LIN {X 0,Y 119.717,Z 305.18,A -85,B 0,C 180,E1 -30603.649,E2 -30603.649} C_VEL
LIN {X 0,Y 116.126,Z 315.063,A -85,B 0,C 180,E1 -30603.943,E2 -30603.943} C_VEL
LIN {X 0,Y 111.009,Z 325.952,A -85,B 0,C 180,E1 -30604.349,E2 -30604.349} C_VEL
LIN {X 0,Y 105.794,Z 334.941,A -85,B 0,C 180,E1 -30604.827,E2 -30604.827} C_VEL
LIN {X 0,Y 99.722,Z 343.662,A -85,B 0,C 180,E1 -30605.461,E2 -30605.461} C_VEL
LIN {X 0,Y 93.661,Z 351.048,A -85,B 0,C 180,E1 -30606.163,E2 -30606.163} C_VEL
LIN {X 0,Y 86.76,Z 358.26,A -85,B 0,C 180,E1 -30607.115,E2 -30607.115} C_VEL
LIN {X 0,Y 79.892,Z 364.456,A -85,B 0,C 180,E1 -30608.255,E2 -30608.255} C_VEL
LIN {X 0,Y 71.375,Z 370.99,A -85,B 0,C 180,E1 -30610.054,E2 -30610.054} C_VEL
LIN {X 0,Y 64.619,Z 375.489,A -85,B 0,C 180,E1 -30611.811,E2 -30611.811} C_VEL
LIN {X 0,Y 54.695,Z 380.985,A -85,B 0,C 180,E1 -30615.484,E2 -30615.484} C_VEL
LIN {X 0,Y 45.01,Z 385.31,A -85,B 0,C 180,E1 -30620.47,E2 -30620.47} C_VEL
LIN {X 0,Y 38.837,Z 387.682,A -85,B 0,C 180,E1 -30625.205,E2 -30625.205} C_VEL
LIN {X 0,Y 32.984,Z 389.485,A -85,B 0,C 180,E1 -30631.54,E2 -30631.54} C_VEL
LIN {X 0,Y 23.511,Z 391.952,A -85,B 0,C 180,E1 -30653.284,E2 -30653.284} C_VEL
LIN {X 0,Y 20.752,Z 392.553,A -85,B 0,C 180,E1 -30670.204,E2 -30670.204} C_VEL
LIN {X 0,Y 19.969,Z 392.717,A -85,B 0,C 180,E1 -30690,E2 -30690} C_VEL
LIN {X 0,Y 20.693,Z 392.552,A -85,B 0,C 180,E1 -30709.854,E2 -30709.854} C_VEL
LIN {X 0,Y 23.498,Z 391.951,A -85,B 0,C 180,E1 -30726.739,E2 -30726.739} C_VEL
LIN {X 0,Y 32.981,Z 389.485,A -85,B 0,C 180,E1 -30748.468,E2 -30748.468} C_VEL
LIN {X 0,Y 41.901,Z 386.53,A -85,B 0,C 180,E1 -30757.293,E2 -30757.293} C_VEL
LIN {X 0,Y 51.443,Z 382.54,A -85,B 0,C 180,E1 -30763,E2 -30763} C_VEL
LIN {X 0,Y 60.969,Z 377.599,A -85,B 0,C 180,E1 -30766.915,E2 -30766.915} C_VEL
LIN {X 0,Y 69.682,Z 372.145,A -85,B 0,C 180,E1 -30769.533,E2 -30769.533} C_VEL
LIN {X 0,Y 78.182,Z 365.831,A -85,B 0,C 180,E1 -30771.422,E2 -30771.422} C_VEL
LIN {X 0,Y 85.041,Z 359.886,A -85,B 0,C 180,E1 -30772.61,E2 -30772.61} C_VEL
LIN {X 0,Y 91.927,Z 352.964,A -85,B 0,C 180,E1 -30773.652,E2 -30773.652} C_VEL
LIN {X 0,Y 98.848,Z 344.794,A -85,B 0,C 180,E1 -30774.487,E2 -30774.487} C_VEL
LIN {X 0,Y 104.925,Z 336.291,A -85,B 0,C 180,E1 -30775.094,E2 -30775.094} C_VEL
LIN {X 0,Y 110.138,Z 327.582,A -85,B 0,C 180,E1 -30775.587,E2 -30775.587} C_VEL
LIN {X 0,Y 114.838,Z 318.036,A -85,B 0,C 180,E1 -30775.963,E2 -30775.963} C_VEL
LIN {X 0,Y 118.374,Z 309.139,A -85,B 0,C 180,E1 -30776.272,E2 -30776.272} C_VEL
LIN {X 0,Y 119.713,Z 305.178,A -85,B 0,C 180,E1 -30776.385,E2 -30776.385} C_VEL
LIN {X 0,Y 120.248,Z 303.503,A -85,B 0,C 180,E1 -30776.648,E2 -30776.648} C_VEL
LIN {X 0,Y 120.44,Z 302.029,A -85,B 0,C 180,E1 -30779.998,E2 -30779.998} C_VEL
LIN {X 0,Y 120.194,Z 303.28,A -85,B 0,C 180,E1 -30783.35,E2 -30783.35} C_VEL
LIN {X 0,Y 120.067,Z 305.276,A -85,B 0,C 180,E1 -30786.721,E2 -30786.721} C_VEL
LIN {X 0,Y 120.02,Z 306.688,A -85,B 0,C 180,E1 -30788.416,E2 -30788.416} C_VEL
LIN {X 0,Y 119.884,Z 309.705,A -85,B 0,C 180,E1 -30791.086,E2 -30791.086} C_VEL
LIN {X 0,Y 119.455,Z 313.518,A -85,B 0,C 180,E1 -30793.609,E2 -30793.609} C_VEL
LIN {X 0,Y 118.463,Z 318.955,A -85,B 0,C 180,E1 -30796.366,E2 -30796.366} C_VEL
LIN {X 0,Y 115.432,Z 330.435,A -85,B 0,C 180,E1 -30801.424,E2 -30801.424} C_VEL
LIN {X 0,Y 112.841,Z 339.939,A -85,B 0,C 180,E1 -30806.593,E2 -30806.593} C_VEL
LIN {X 0,Y 110.853,Z 348.799,A -85,B 0,C 180,E1 -30812.532,E2 -30812.532} C_VEL
LIN {X 0,Y 109.913,Z 356.079,A -85,B 0,C 180,E1 -30818.394,E2 -30818.394} C_VEL
LIN {X 0,Y 110.102,Z 362.578,A -85,B 0,C 180,E1 -30824.597,E2 -30824.597} C_VEL
LIN {X 0,Y 111.723,Z 368.309,A -85,B 0,C 180,E1 -30831.02,E2 -30831.02} C_VEL
LIN {X 0,Y 115.499,Z 373.969,A -85,B 0,C 180,E1 -30838.413,E2 -30838.413} C_VEL
LIN {X 0,Y 120.451,Z 378.02,A -85,B 0,C 180,E1 -30844.486,E2 -30844.486} C_VEL
LIN {X 0,Y 127.757,Z 381.631,A -85,B 0,C 180,E1 -30850.727,E2 -30850.727} C_VEL
LIN {X 0,Y 137.278,Z 384.47,A -85,B 0,C 180,E1 -30856.578,E2 -30856.578} C_VEL
LIN {X 0,Y 149.17,Z 386.419,A -85,B 0,C 180,E1 -30861.875,E2 -30861.875} C_VEL
LIN {X 0,Y 161.996,Z 387.374,A -85,B 0,C 180,E1 -30866.197,E2 -30866.197} C_VEL
LIN {X 0,Y 176.187,Z 387.451,A -85,B 0,C 180,E1 -30870,E2 -30870} C_VEL
LIN {X 0,Y 161.994,Z 387.377,A -85,B 0,C 180,E1 -30873.788,E2 -30873.788} C_VEL
LIN {X 0,Y 156.857,Z 387.171,A -85,B 0,C 180,E1 -30875.379,E2 -30875.379} C_VEL
LIN {X 0,Y 152.092,Z 386.947,A -85,B 0,C 180,E1 -30876.675,E2 -30876.675} C_VEL
LIN {X 0,Y 136.433,Z 386.309,A -85,B 0,C 180,E1 -30880.073,E2 -30880.073} C_VEL
LIN {X 0,Y 131.842,Z 385.916,A -85,B 0,C 180,E1 -30881.644,E2 -30881.644} C_VEL
LIN {X 0,Y 130.521,Z 385.655,A -85,B 0,C 180,E1 -30882.275,E2 -30882.275} C_VEL
LIN {X 0,Y 123.482,Z 384.041,A -85,B 0,C 180,E1 -30886.533,E2 -30886.533} C_VEL
LIN {X 0,Y 114.992,Z 380.706,A -85,B 0,C 180,E1 -30893.549,E2 -30893.549} C_VEL
LIN {X 0,Y 108.159,Z 375.569,A -85,B 0,C 180,E1 -30902.362,E2 -30902.362} C_VEL
LIN {X 0,Y 104.996,Z 370.6,A -85,B 0,C 180,E1 -30909.671,E2 -30909.671} C_VEL
LIN {X 0,Y 103.683,Z 364.458,A -85,B 0,C 180,E1 -30917.328,E2 -30917.328} C_VEL
LIN {X 0,Y 104.187,Z 357.94,A -85,B 0,C 180,E1 -30924.043,E2 -30924.043} C_VEL
LIN {X 0,Y 105.674,Z 351.257,A -85,B 0,C 180,E1 -30929.834,E2 -30929.834} C_VEL
LIN {X 0,Y 108.139,Z 343.326,A -85,B 0,C 180,E1 -30935.485,E2 -30935.485} C_VEL
LIN {X 0,Y 110.828,Z 335.561,A -85,B 0,C 180,E1 -30940.076,E2 -30940.076} C_VEL
LIN {X 0,Y 114.078,Z 326.223,A -85,B 0,C 180,E1 -30944.597,E2 -30944.597} C_VEL
LIN {X 0,Y 116.107,Z 319.796,A -85,B 0,C 180,E1 -30947.593,E2 -30947.593} C_VEL
LIN {X 0,Y 117.011,Z 315.348,A -85,B 0,C 180,E1 -30950.495,E2 -30950.495} C_VEL
LIN {X 0,Y 117.648,Z 311.793,A -85,B 0,C 180,E1 -30954.051,E2 -30954.051} C_VEL
LIN {X 0,Y 117.816,Z 310.254,A -85,B 0,C 180,E1 -30956.582,E2 -30956.582} C_VEL
LIN {X 0,Y 118.131,Z 308.908,A -85,B 0,C 180,E1 -30960.002,E2 -30960.002} C_VEL
LIN {X 0,Y 117.855,Z 309.739,A -85,B 0,C 180,E1 -30960.319,E2 -30960.319} C_VEL
LIN {X 0,Y 112.453,Z 322.497,A -85,B 0,C 180,E1 -30960.592,E2 -30960.592} C_VEL
LIN {X 0,Y 106.311,Z 333.399,A -85,B 0,C 180,E1 -30960.926,E2 -30960.926} C_VEL
LIN {X 0,Y 100.174,Z 342.337,A -85,B 0,C 180,E1 -30961.31,E2 -30961.31} C_VEL
LIN {X 0,Y 93.166,Z 350.856,A -85,B 0,C 180,E1 -30961.801,E2 -30961.801} C_VEL
LIN {X 0,Y 86.169,Z 358.068,A -85,B 0,C 180,E1 -30962.416,E2 -30962.416} C_VEL
LIN {X 0,Y 79.183,Z 364.264,A -85,B 0,C 180,E1 -30963.146,E2 -30963.146} C_VEL
LIN {X 0,Y 70.481,Z 370.797,A -85,B 0,C 180,E1 -30964.337,E2 -30964.337} C_VEL
LIN {X 0,Y 63.544,Z 375.296,A -85,B 0,C 180,E1 -30965.506,E2 -30965.506} C_VEL
LIN {X 0,Y 54.523,Z 380.204,A -85,B 0,C 180,E1 -30967.657,E2 -30967.657} C_VEL
LIN {X 0,Y 46.422,Z 383.878,A -85,B 0,C 180,E1 -30970.249,E2 -30970.249} C_VEL
LIN {X 0,Y 36.38,Z 387.49,A -85,B 0,C 180,E1 -30975.003,E2 -30975.003} C_VEL
LIN {X 0,Y 29.879,Z 389.292,A -85,B 0,C 180,E1 -30979.807,E2 -30979.807} C_VEL
LIN {X 0,Y 18.307,Z 391.76,A -85,B 0,C 180,E1 -30999.844,E2 -30999.844} C_VEL
LIN {X 0,Y 14.255,Z 392.361,A -85,B 0,C 180,E1 -31020.461,E2 -31020.461} C_VEL
LIN {X 0,Y 12.863,Z 392.526,A -85,B 0,C 180,E1 -31050,E2 -31050} C_VEL
LIN {X 0,Y 14.211,Z 392.36,A -85,B 0,C 180,E1 -31079.64,E2 -31079.64} C_VEL
LIN {X 0,Y 18.298,Z 391.759,A -85,B 0,C 180,E1 -31100.189,E2 -31100.189} C_VEL
LIN {X 0,Y 29.878,Z 389.292,A -85,B 0,C 180,E1 -31120.201,E2 -31120.201} C_VEL
LIN {X 0,Y 39.698,Z 386.338,A -85,B 0,C 180,E1 -31126.825,E2 -31126.825} C_VEL
LIN {X 0,Y 49.826,Z 382.347,A -85,B 0,C 180,E1 -31130.877,E2 -31130.877} C_VEL
LIN {X 0,Y 56.661,Z 379.131,A -85,B 0,C 180,E1 -31132.871,E2 -31132.871} C_VEL
LIN {X 0,Y 67.01,Z 373.107,A -85,B 0,C 180,E1 -31135.098,E2 -31135.098} C_VEL
LIN {X 0,Y 75.698,Z 367.014,A -85,B 0,C 180,E1 -31136.42,E2 -31136.42} C_VEL
LIN {X 0,Y 82.675,Z 361.319,A -85,B 0,C 180,E1 -31137.231,E2 -31137.231} C_VEL
LIN {X 0,Y 91.414,Z 352.772,A -85,B 0,C 180,E1 -31138.084,E2 -31138.084} C_VEL
LIN {X 0,Y 98.42,Z 344.602,A -85,B 0,C 180,E1 -31138.601,E2 -31138.601} C_VEL
LIN {X 0,Y 104.557,Z 336.1,A -85,B 0,C 180,E1 -31138.968,E2 -31138.968} C_VEL
LIN {X 0,Y 109.82,Z 327.39,A -85,B 0,C 180,E1 -31139.289,E2 -31139.289} C_VEL
LIN {X 0,Y 114.558,Z 317.844,A -85,B 0,C 180,E1 -31139.51,E2 -31139.51} C_VEL
LIN {X 0,Y 117.855,Z 309.739,A -85,B 0,C 180,E1 -31139.689,E2 -31139.689} C_VEL
LIN {X 0,Y 118.131,Z 308.909,A -85,B 0,C 180,E1 -31139.998,E2 -31139.998} C_VEL
LIN {X 0,Y 117.815,Z 310.257,A -85,B 0,C 180,E1 -31143.418,E2 -31143.418} C_VEL
LIN {X 0,Y 117.528,Z 312.556,A -85,B 0,C 180,E1 -31146.867,E2 -31146.867} C_VEL
LIN {X 0,Y 117.015,Z 315.34,A -85,B 0,C 180,E1 -31149.505,E2 -31149.505} C_VEL
LIN {X 0,Y 116.112,Z 319.784,A -85,B 0,C 180,E1 -31152.406,E2 -31152.406} C_VEL
LIN {X 0,Y 114.581,Z 324.734,A -85,B 0,C 180,E1 -31154.762,E2 -31154.762} C_VEL
LIN {X 0,Y 111.471,Z 333.723,A -85,B 0,C 180,E1 -31158.966,E2 -31158.966} C_VEL
LIN {X 0,Y 109.082,Z 340.55,A -85,B 0,C 180,E1 -31162.739,E2 -31162.739} C_VEL
LIN {X 0,Y 106.334,Z 349.039,A -85,B 0,C 180,E1 -31168.488,E2 -31168.488} C_VEL
LIN {X 0,Y 104.477,Z 356.334,A -85,B 0,C 180,E1 -31174.467,E2 -31174.467} C_VEL
LIN {X 0,Y 103.688,Z 362.492,A -85,B 0,C 180,E1 -31180.491,E2 -31180.491} C_VEL
LIN {X 0,Y 104.337,Z 368.701,A -85,B 0,C 180,E1 -31187.809,E2 -31187.809} C_VEL
LIN {X 0,Y 106.893,Z 374.031,A -85,B 0,C 180,E1 -31195.263,E2 -31195.263} C_VEL
LIN {X 0,Y 111.223,Z 378.305,A -85,B 0,C 180,E1 -31202.203,E2 -31202.203} C_VEL
LIN {X 0,Y 117.698,Z 381.92,A -85,B 0,C 180,E1 -31209.006,E2 -31209.006} C_VEL
LIN {X 0,Y 124.291,Z 384.232,A -85,B 0,C 180,E1 -31213.992,E2 -31213.992} C_VEL
LIN {X 0,Y 135.506,Z 386.463,A -85,B 0,C 180,E1 -31220.197,E2 -31220.197} C_VEL
LIN {X 0,Y 148.1,Z 387.613,A -85,B 0,C 180,E1 -31225.215,E2 -31225.215} C_VEL
LIN {X 0,Y 164.229,Z 387.768,A -85,B 0,C 180,E1 -31230,E2 -31230} C_VEL
LIN {X 0,Y 148.095,Z 387.618,A -85,B 0,C 180,E1 -31234.764,E2 -31234.764} C_VEL
LIN {X 0,Y 135.506,Z 386.463,A -85,B 0,C 180,E1 -31239.803,E2 -31239.803} C_VEL
LIN {X 0,Y 130.521,Z 385.655,A -85,B 0,C 180,E1 -31242.275,E2 -31242.275} C_VEL
LIN {X 0,Y 126.383,Z 385.107,A -85,B 0,C 180,E1 -31244.144,E2 -31244.144} C_VEL
LIN {X 0,Y 112.702,Z 383.535,A -85,B 0,C 180,E1 -31249.585,E2 -31249.585} C_VEL
LIN {X 0,Y 109.04,Z 382.656,A -85,B 0,C 180,E1 -31251.925,E2 -31251.925} C_VEL
LIN {X 0,Y 108.082,Z 382.289,A -85,B 0,C 180,E1 -31252.809,E2 -31252.809} C_VEL
LIN {X 0,Y 103.628,Z 379.673,A -85,B 0,C 180,E1 -31258.342,E2 -31258.342} C_VEL
LIN {X 0,Y 99.538,Z 375.349,A -85,B 0,C 180,E1 -31266.247,E2 -31266.247} C_VEL
LIN {X 0,Y 97.636,Z 370.393,A -85,B 0,C 180,E1 -31273.964,E2 -31273.964} C_VEL
LIN {X 0,Y 97.46,Z 366.272,A -85,B 0,C 180,E1 -31279.536,E2 -31279.536} C_VEL
LIN {X 0,Y 98.847,Z 359.058,A -85,B 0,C 180,E1 -31287.491,E2 -31287.491} C_VEL
LIN {X 0,Y 100.988,Z 352.866,A -85,B 0,C 180,E1 -31293.11,E2 -31293.11} C_VEL
LIN {X 0,Y 104.52,Z 344.31,A -85,B 0,C 180,E1 -31299.333,E2 -31299.333} C_VEL
LIN {X 0,Y 108.138,Z 335.987,A -85,B 0,C 180,E1 -31304.221,E2 -31304.221} C_VEL
LIN {X 0,Y 111.793,Z 327.342,A -85,B 0,C 180,E1 -31308.347,E2 -31308.347} C_VEL
LIN {X 0,Y 113.197,Z 323.573,A -85,B 0,C 180,E1 -31310.282,E2 -31310.282} C_VEL
LIN {X 0,Y 114.321,Z 319.955,A -85,B 0,C 180,E1 -31312.939,E2 -31312.939} C_VEL
LIN {X 0,Y 114.743,Z 318.21,A -85,B 0,C 180,E1 -31314.73,E2 -31314.73} C_VEL
LIN {X 0,Y 114.98,Z 317.143,A -85,B 0,C 180,E1 -31316.498,E2 -31316.498} C_VEL
LIN {X 0,Y 114.32,Z 318.561,A -85,B 0,C 180,E1 -31316.943,E2 -31316.943} C_VEL
LIN {X 0,Y 108.198,Z 330.439,A -85,B 0,C 180,E1 -31317.047,E2 -31317.047} C_VEL
LIN {X 0,Y 101.146,Z 341.011,A -85,B 0,C 180,E1 -31317.218,E2 -31317.218} C_VEL
LIN {X 0,Y 94.977,Z 348.747,A -85,B 0,C 180,E1 -31317.371,E2 -31317.371} C_VEL
LIN {X 0,Y 86.162,Z 357.876,A -85,B 0,C 180,E1 -31317.688,E2 -31317.688} C_VEL
LIN {X 0,Y 79.113,Z 364.072,A -85,B 0,C 180,E1 -31317.991,E2 -31317.991} C_VEL
LIN {X 0,Y 70.302,Z 370.605,A -85,B 0,C 180,E1 -31318.541,E2 -31318.541} C_VEL
LIN {X 0,Y 63.26,Z 375.104,A -85,B 0,C 180,E1 -31319.06,E2 -31319.06} C_VEL
LIN {X 0,Y 53.07,Z 380.439,A -85,B 0,C 180,E1 -31320.253,E2 -31320.253} C_VEL
LIN {X 0,Y 42.194,Z 384.926,A -85,B 0,C 180,E1 -31322.012,E2 -31322.012} C_VEL
LIN {X 0,Y 35.215,Z 387.298,A -85,B 0,C 180,E1 -31323.744,E2 -31323.744} C_VEL
LIN {X 0,Y 28.272,Z 389.1,A -85,B 0,C 180,E1 -31326.096,E2 -31326.096} C_VEL
LIN {X 0,Y 14.789,Z 391.567,A -85,B 0,C 180,E1 -31338.122,E2 -31338.122} C_VEL
LIN {X 0,Y 8.797,Z 392.169,A -85,B 0,C 180,E1 -31356.976,E2 -31356.976} C_VEL
LIN {X 0,Y 5.749,Z 392.334,A -85,B 0,C 180,E1 -31410,E2 -31410} C_VEL
LIN {X 0,Y 8.772,Z 392.168,A -85,B 0,C 180,E1 -31463.24,E2 -31463.24} C_VEL
LIN {X 0,Y 14.786,Z 391.567,A -85,B 0,C 180,E1 -31481.923,E2 -31481.923} C_VEL
LIN {X 0,Y 28.271,Z 389.1,A -85,B 0,C 180,E1 -31493.912,E2 -31493.912} C_VEL
LIN {X 0,Y 38.701,Z 386.145,A -85,B 0,C 180,E1 -31497.174,E2 -31497.174} C_VEL
LIN {X 0,Y 49.201,Z 382.155,A -85,B 0,C 180,E1 -31499.113,E2 -31499.113} C_VEL
LIN {X 0,Y 56.223,Z 378.938,A -85,B 0,C 180,E1 -31500.109,E2 -31500.109} C_VEL
LIN {X 0,Y 66.78,Z 372.915,A -85,B 0,C 180,E1 -31501.195,E2 -31501.195} C_VEL
LIN {X 0,Y 75.588,Z 366.822,A -85,B 0,C 180,E1 -31501.819,E2 -31501.819} C_VEL
LIN {X 0,Y 82.637,Z 361.127,A -85,B 0,C 180,E1 -31502.16,E2 -31502.16} C_VEL
LIN {X 0,Y 91.453,Z 352.58,A -85,B 0,C 180,E1 -31502.542,E2 -31502.542} C_VEL
LIN {X 0,Y 98.503,Z 344.411,A -85,B 0,C 180,E1 -31502.731,E2 -31502.731} C_VEL
LIN {X 0,Y 104.67,Z 335.908,A -85,B 0,C 180,E1 -31502.852,E2 -31502.852} C_VEL
LIN {X 0,Y 109.73,Z 327.624,A -85,B 0,C 180,E1 -31502.981,E2 -31502.981} C_VEL
LIN {X 0,Y 114.154,Z 318.938,A -85,B 0,C 180,E1 -31503.048,E2 -31503.048} C_VEL
LIN {X 0,Y 114.977,Z 317.151,A -85,B 0,C 180,E1 -31503.502,E2 -31503.502} C_VEL
LIN {X 0,Y 114.73,Z 318.239,A -85,B 0,C 180,E1 -31505.27,E2 -31505.27} C_VEL
LIN {X 0,Y 114.07,Z 320.946,A -85,B 0,C 180,E1 -31507.878,E2 -31507.878} C_VEL
LIN {X 0,Y 113.191,Z 323.583,A -85,B 0,C 180,E1 -31509.718,E2 -31509.718} C_VEL
LIN {X 0,Y 111.794,Z 327.348,A -85,B 0,C 180,E1 -31511.664,E2 -31511.664} C_VEL
LIN {X 0,Y 107.515,Z 337.525,A -85,B 0,C 180,E1 -31516.593,E2 -31516.593} C_VEL
LIN {X 0,Y 103.001,Z 347.918,A -85,B 0,C 180,E1 -31523.097,E2 -31523.097} C_VEL
LIN {X 0,Y 99.626,Z 356.578,A -85,B 0,C 180,E1 -31530.163,E2 -31530.163} C_VEL
LIN {X 0,Y 97.918,Z 362.751,A -85,B 0,C 180,E1 -31536.37,E2 -31536.37} C_VEL
LIN {X 0,Y 97.425,Z 368.832,A -85,B 0,C 180,E1 -31543.832,E2 -31543.832} C_VEL
LIN {X 0,Y 98.753,Z 374.021,A -85,B 0,C 180,E1 -31551.518,E2 -31551.518} C_VEL
LIN {X 0,Y 102.11,Z 378.453,A -85,B 0,C 180,E1 -31559.266,E2 -31559.266} C_VEL
LIN {X 0,Y 107.875,Z 382.206,A -85,B 0,C 180,E1 -31566.99,E2 -31566.99} C_VEL
LIN {X 0,Y 113.233,Z 384.33,A -85,B 0,C 180,E1 -31571.921,E2 -31571.921} C_VEL
LIN {X 0,Y 122.133,Z 386.449,A -85,B 0,C 180,E1 -31578.018,E2 -31578.018} C_VEL
LIN {X 0,Y 134.476,Z 387.839,A -85,B 0,C 180,E1 -31584,E2 -31584} C_VEL
LIN {X 0,Y 147.626,Z 388.209,A -85,B 0,C 180,E1 -31588.622,E2 -31588.622} C_VEL
LIN {X 0,Y 152.296,Z 388.084,A -85,B 0,C 180,E1 -31590,E2 -31590} C_VEL
LIN {X 0,Y 140.828,Z 388.098,A -85,B 0,C 180,E1 -31593.564,E2 -31593.564} C_VEL
LIN {X 0,Y 128.019,Z 387.219,A -85,B 0,C 180,E1 -31598.836,E2 -31598.836} C_VEL
LIN {X 0,Y 119.391,Z 385.888,A -85,B 0,C 180,E1 -31603.619,E2 -31603.619} C_VEL
LIN {X 0,Y 111.723,Z 383.815,A -85,B 0,C 180,E1 -31609.344,E2 -31609.344} C_VEL
LIN {X 0,Y 108.082,Z 382.289,A -85,B 0,C 180,E1 -31612.809,E2 -31612.809} C_VEL
LIN {X 0,Y 105.046,Z 381.281,A -85,B 0,C 180,E1 -31615.486,E2 -31615.486} C_VEL
LIN {X 0,Y 94.843,Z 378.641,A -85,B 0,C 180,E1 -31623.749,E2 -31623.749} C_VEL
LIN {X 0,Y 92.636,Z 377.218,A -85,B 0,C 180,E1 -31626.968,E2 -31626.968} C_VEL
LIN {X 0,Y 92.209,Z 376.621,A -85,B 0,C 180,E1 -31628.096,E2 -31628.096} C_VEL
LIN {X 0,Y 91.002,Z 372.12,A -85,B 0,C 180,E1 -31635.971,E2 -31635.971} C_VEL
LIN {X 0,Y 91.937,Z 365.634,A -85,B 0,C 180,E1 -31645.023,E2 -31645.023} C_VEL
LIN {X 0,Y 94.304,Z 359.218,A -85,B 0,C 180,E1 -31652.244,E2 -31652.244} C_VEL
LIN {X 0,Y 97.979,Z 351.735,A -85,B 0,C 180,E1 -31658.824,E2 -31658.824} C_VEL
LIN {X 0,Y 102.175,Z 343.794,A -85,B 0,C 180,E1 -31664.357,E2 -31664.357} C_VEL
LIN {X 0,Y 106.125,Z 336.294,A -85,B 0,C 180,E1 -31668.543,E2 -31668.543} C_VEL
LIN {X 0,Y 109.814,Z 328.832,A -85,B 0,C 180,E1 -31672.195,E2 -31672.195} C_VEL
LIN {X 0,Y 110.156,Z 328.004,A -85,B 0,C 180,E1 -31672.671,E2 -31672.671} C_VEL
LIN {X 0,Y 109.108,Z 329.688,A -85,B 0,C 180,E1 -31673.32,E2 -31673.32} C_VEL
LIN {X 0,Y 101.739,Z 340.819,A -85,B 0,C 180,E1 -31673.215,E2 -31673.215} C_VEL
LIN {X 0,Y 95.565,Z 348.556,A -85,B 0,C 180,E1 -31673.121,E2 -31673.121} C_VEL
LIN {X 0,Y 86.741,Z 357.685,A -85,B 0,C 180,E1 -31672.988,E2 -31672.988} C_VEL
LIN {X 0,Y 79.682,Z 363.879,A -85,B 0,C 180,E1 -31672.862,E2 -31672.862} C_VEL
LIN {X 0,Y 70.844,Z 370.412,A -85,B 0,C 180,E1 -31672.759,E2 -31672.759} C_VEL
LIN {X 0,Y 63.775,Z 374.912,A -85,B 0,C 180,E1 -31672.652,E2 -31672.652} C_VEL
LIN {X 0,Y 52.528,Z 380.681,A -85,B 0,C 180,E1 -31672.569,E2 -31672.569} C_VEL
LIN {X 0,Y 42.543,Z 384.734,A -85,B 0,C 180,E1 -31672.384,E2 -31672.384} C_VEL
LIN {X 0,Y 35.468,Z 387.105,A -85,B 0,C 180,E1 -31672.192,E2 -31672.192} C_VEL
LIN {X 0,Y 28.411,Z 388.908,A -85,B 0,C 180,E1 -31671.673,E2 -31671.673} C_VEL
LIN {X 0,Y 14.284,Z 391.375,A -85,B 0,C 180,E1 -31669.74,E2 -31669.74} C_VEL
LIN {X 0,Y 7.265,Z 391.977,A -85,B 0,C 180,E1 -31665.323,E2 -31665.323} C_VEL
LIN {X 0,Y 1.35,Z 392.142,A -85,B 0,C 180,E1 -31590,E2 -31590} C_VEL
LIN {X 0,Y 7.274,Z 391.976,A -85,B 0,C 180,E1 -31514.953,E2 -31514.953} C_VEL
LIN {X 0,Y 14.286,Z 391.374,A -85,B 0,C 180,E1 -31510.308,E2 -31510.308} C_VEL
LIN {X 0,Y 28.412,Z 388.908,A -85,B 0,C 180,E1 -31508.334,E2 -31508.334} C_VEL
LIN {X 0,Y 39.007,Z 385.952,A -85,B 0,C 180,E1 -31507.723,E2 -31507.723} C_VEL
LIN {X 0,Y 49.607,Z 381.962,A -85,B 0,C 180,E1 -31507.386,E2 -31507.386} C_VEL
LIN {X 0,Y 56.686,Z 378.746,A -85,B 0,C 180,E1 -31507.326,E2 -31507.326} C_VEL
LIN {X 0,Y 67.307,Z 372.723,A -85,B 0,C 180,E1 -31507.272,E2 -31507.272} C_VEL
LIN {X 0,Y 76.147,Z 366.63,A -85,B 0,C 180,E1 -31507.181,E2 -31507.181} C_VEL
LIN {X 0,Y 83.208,Z 360.935,A -85,B 0,C 180,E1 -31507.057,E2 -31507.057} C_VEL
LIN {X 0,Y 92.043,Z 352.388,A -85,B 0,C 180,E1 -31506.967,E2 -31506.967} C_VEL
LIN {X 0,Y 99.095,Z 344.219,A -85,B 0,C 180,E1 -31506.832,E2 -31506.832} C_VEL
LIN {X 0,Y 105.262,Z 335.717,A -85,B 0,C 180,E1 -31506.714,E2 -31506.714} C_VEL
LIN {X 0,Y 109.111,Z 329.682,A -85,B 0,C 180,E1 -31506.68,E2 -31506.68} C_VEL
LIN {X 0,Y 110.169,Z 327.98,A -85,B 0,C 180,E1 -31507.328,E2 -31507.328} C_VEL
LIN {X 0,Y 108.09,Z 332.431,A -85,B 0,C 180,E1 -31509.585,E2 -31509.585} C_VEL
LIN {X 0,Y 103.81,Z 340.756,A -85,B 0,C 180,E1 -31513.814,E2 -31513.814} C_VEL
LIN {X 0,Y 99.099,Z 349.573,A -85,B 0,C 180,E1 -31519.518,E2 -31519.518} C_VEL
LIN {X 0,Y 95.415,Z 356.863,A -85,B 0,C 180,E1 -31525.544,E2 -31525.544} C_VEL
LIN {X 0,Y 92.705,Z 363.199,A -85,B 0,C 180,E1 -31532.048,E2 -31532.048} C_VEL
LIN {X 0,Y 91.098,Z 369.089,A -85,B 0,C 180,E1 -31539.514,E2 -31539.514} C_VEL
LIN {X 0,Y 91.275,Z 374.177,A -85,B 0,C 180,E1 -31547.501,E2 -31547.501} C_VEL
LIN {X 0,Y 93.465,Z 378.582,A -85,B 0,C 180,E1 -31555.801,E2 -31555.801} C_VEL
LIN {X 0,Y 98.43,Z 382.485,A -85,B 0,C 180,E1 -31564.634,E2 -31564.634} C_VEL
LIN {X 0,Y 104.076,Z 384.887,A -85,B 0,C 180,E1 -31570.969,E2 -31570.969} C_VEL
LIN {X 0,Y 114.583,Z 387.2,A -85,B 0,C 180,E1 -31578.911,E2 -31578.911} C_VEL
LIN {X 0,Y 123.062,Z 388.144,A -85,B 0,C 180,E1 -31583.442,E2 -31583.442} C_VEL
LIN {X 0,Y 133.633,Z 388.548,A -85,B 0,C 180,E1 -31587.723,E2 -31587.723} C_VEL
LIN {X 0,Y 140.418,Z 388.398,A -85,B 0,C 180,E1 -31590,E2 -31590} C_VEL
LIN {X 0,Y 126.954,Z 388.307,A -85,B 0,C 180,E1 -31594.85,E2 -31594.85} C_VEL
LIN {X 0,Y 115.539,Z 387.328,A -85,B 0,C 180,E1 -31600.514,E2 -31600.514} C_VEL
LIN {X 0,Y 108.852,Z 386.181,A -85,B 0,C 180,E1 -31604.967,E2 -31604.967} C_VEL
LIN {X 0,Y 101.85,Z 384.071,A -85,B 0,C 180,E1 -31611.281,E2 -31611.281} C_VEL
LIN {X 0,Y 96.204,Z 381.129,A -85,B 0,C 180,E1 -31618.765,E2 -31618.765} C_VEL
LIN {X 0,Y 92.209,Z 376.621,A -85,B 0,C 180,E1 -31628.096,E2 -31628.096} C_VEL
LIN {X 0,Y 90.813,Z 374.958,A -85,B 0,C 180,E1 -31631.533,E2 -31631.533} C_VEL
LIN {X 0,Y 86.018,Z 370.75,A -85,B 0,C 180,E1 -31642.321,E2 -31642.321} C_VEL
LIN {X 0,Y 85.83,Z 368.79,A -85,B 0,C 180,E1 -31646.016,E2 -31646.016} C_VEL
LIN {X 0,Y 86.075,Z 368.012,A -85,B 0,C 180,E1 -31647.204,E2 -31647.204} C_VEL
LIN {X 0,Y 89.354,Z 361.507,A -85,B 0,C 180,E1 -31655.215,E2 -31655.215} C_VEL
LIN {X 0,Y 94.335,Z 353.36,A -85,B 0,C 180,E1 -31662.665,E2 -31662.665} C_VEL
LIN {X 0,Y 99.436,Z 345.305,A -85,B 0,C 180,E1 -31668.306,E2 -31668.306} C_VEL
LIN {X 0,Y 100.182,Z 344.028,A -85,B 0,C 180,E1 -31669.149,E2 -31669.149} C_VEL
LIN {X 0,Y 93.169,Z 352.197,A -85,B 0,C 180,E1 -31668.701,E2 -31668.701} C_VEL
LIN {X 0,Y 84.383,Z 360.743,A -85,B 0,C 180,E1 -31668.127,E2 -31668.127} C_VEL
LIN {X 0,Y 73.843,Z 369.065,A -85,B 0,C 180,E1 -31667.298,E2 -31667.298} C_VEL
LIN {X 0,Y 65.071,Z 374.719,A -85,B 0,C 180,E1 -31666.416,E2 -31666.416} C_VEL
LIN {X 0,Y 54.975,Z 380.018,A -85,B 0,C 180,E1 -31665.19,E2 -31665.19} C_VEL
LIN {X 0,Y 47.521,Z 383.301,A -85,B 0,C 180,E1 -31664.005,E2 -31664.005} C_VEL
LIN {X 0,Y 37.118,Z 386.913,A -85,B 0,C 180,E1 -31661.207,E2 -31661.207} C_VEL
LIN {X 0,Y 23.547,Z 390.111,A -85,B 0,C 180,E1 -31653.559,E2 -31653.559} C_VEL
LIN {X 0,Y 17.068,Z 391.182,A -85,B 0,C 180,E1 -31645.44,E2 -31645.44} C_VEL
LIN {X 0,Y 11.391,Z 391.784,A -85,B 0,C 180,E1 -31628.095,E2 -31628.095} C_VEL
LIN {X 0,Y 8.44,Z 391.951,A -85,B 0,C 180,E1 -31590,E2 -31590} C_VEL
LIN {X 0,Y 11.415,Z 391.784,A -85,B 0,C 180,E1 -31551.998,E2 -31551.998} C_VEL
LIN {X 0,Y 17.074,Z 391.182,A -85,B 0,C 180,E1 -31534.59,E2 -31534.59} C_VEL
LIN {X 0,Y 30.272,Z 388.716,A -85,B 0,C 180,E1 -31521.775,E2 -31521.775} C_VEL
LIN {X 0,Y 40.589,Z 385.759,A -85,B 0,C 180,E1 -31517.766,E2 -31517.766} C_VEL
LIN {X 0,Y 51.023,Z 381.769,A -85,B 0,C 180,E1 -31515.383,E2 -31515.383} C_VEL
LIN {X 0,Y 61.544,Z 376.637,A -85,B 0,C 180,E1 -31513.916,E2 -31513.916} C_VEL
LIN {X 0,Y 70.329,Z 371.376,A -85,B 0,C 180,E1 -31513.016,E2 -31513.016} C_VEL
LIN {X 0,Y 79.118,Z 365.062,A -85,B 0,C 180,E1 -31512.283,E2 -31512.283} C_VEL
LIN {X 0,Y 86.143,Z 359.117,A -85,B 0,C 180,E1 -31511.759,E2 -31511.759} C_VEL
LIN {X 0,Y 93.172,Z 352.197,A -85,B 0,C 180,E1 -31511.308,E2 -31511.308} C_VEL
LIN {X 0,Y 100.187,Z 344.028,A -85,B 0,C 180,E1 -31510.865,E2 -31510.865} C_VEL
LIN {X 0,Y 94.275,Z 353.429,A -85,B 0,C 180,E1 -31517.347,E2 -31517.347} C_VEL
LIN {X 0,Y 89.36,Z 361.514,A -85,B 0,C 180,E1 -31524.807,E2 -31524.807} C_VEL
LIN {X 0,Y 85.841,Z 368.487,A -85,B 0,C 180,E1 -31533.43,E2 -31533.43} C_VEL
LIN {X 0,Y 84.489,Z 373.713,A -85,B 0,C 180,E1 -31541.714,E2 -31541.714} C_VEL
LIN {X 0,Y 85.329,Z 378.598,A -85,B 0,C 180,E1 -31551.477,E2 -31551.477} C_VEL
LIN {X 0,Y 88.672,Z 382.363,A -85,B 0,C 180,E1 -31560.668,E2 -31560.668} C_VEL
LIN {X 0,Y 93.38,Z 384.901,A -85,B 0,C 180,E1 -31567.895,E2 -31567.895} C_VEL
LIN {X 0,Y 101.461,Z 387.121,A -85,B 0,C 180,E1 -31575.863,E2 -31575.863} C_VEL
LIN {X 0,Y 113.189,Z 388.499,A -85,B 0,C 180,E1 -31583.421,E2 -31583.421} C_VEL
LIN {X 0,Y 126.512,Z 388.767,A -85,B 0,C 180,E1 -31589.19,E2 -31589.19} C_VEL
LIN {X 0,Y 128.789,Z 388.706,A -85,B 0,C 180,E1 -31590,E2 -31590} C_VEL
LIN {X 0,Y 119.693,Z 388.782,A -85,B 0,C 180,E1 -31593.48,E2 -31593.48} C_VEL
LIN {X 0,Y 107.072,Z 387.937,A -85,B 0,C 180,E1 -31600.092,E2 -31600.092} C_VEL
LIN {X 0,Y 98.641,Z 386.467,A -85,B 0,C 180,E1 -31606.558,E2 -31606.558} C_VEL
LIN {X 0,Y 92.13,Z 384.353,A -85,B 0,C 180,E1 -31613.743,E2 -31613.743} C_VEL
LIN {X 0,Y 86.397,Z 380.217,A -85,B 0,C 180,E1 -31624.709,E2 -31624.709} C_VEL
LIN {X 0,Y 84.759,Z 377.125,A -85,B 0,C 180,E1 -31631.737,E2 -31631.737} C_VEL
LIN {X 0,Y 84.803,Z 371.698,A -85,B 0,C 180,E1 -31641.658,E2 -31641.658} C_VEL
LIN {X 0,Y 86.075,Z 368.012,A -85,B 0,C 180,E1 -31647.204,E2 -31647.204} C_VEL
LIN {X 0,Y 86.264,Z 366.612,A -85,B 0,C 180,E1 -31649.695,E2 -31649.695} C_VEL
LIN {X 0,Y 85.17,Z 363.237,A -85,B 0,C 180,E1 -31658.412,E2 -31658.412} C_VEL
LIN {X 0,Y 86.09,Z 361.606,A -85,B 0,C 180,E1 -31660.754,E2 -31660.754} C_VEL
LIN {X 0,Y 88.04,Z 358.909,A -85,B 0,C 180,E1 -31663.32,E2 -31663.32} C_VEL
LIN {X 0,Y 87.871,Z 358.925,A -85,B 0,C 180,E1 -31663.691,E2 -31663.691} C_VEL
LIN {X 0,Y 80.931,Z 364.87,A -85,B 0,C 180,E1 -31662.79,E2 -31662.79} C_VEL
LIN {X 0,Y 72.273,Z 371.183,A -85,B 0,C 180,E1 -31661.461,E2 -31661.461} C_VEL
LIN {X 0,Y 63.662,Z 376.443,A -85,B 0,C 180,E1 -31659.778,E2 -31659.778} C_VEL
LIN {X 0,Y 53.373,Z 381.575,A -85,B 0,C 180,E1 -31657.179,E2 -31657.179} C_VEL
LIN {X 0,Y 43.303,Z 385.567,A -85,B 0,C 180,E1 -31653.205,E2 -31653.205} C_VEL
LIN {X 0,Y 33.563,Z 388.524,A -85,B 0,C 180,E1 -31646.884,E2 -31646.884} C_VEL
LIN {X 0,Y 21.913,Z 390.99,A -85,B 0,C 180,E1 -31629.899,E2 -31629.899} C_VEL
LIN {X 0,Y 17.548,Z 391.592,A -85,B 0,C 180,E1 -31613.609,E2 -31613.609} C_VEL
LIN {X 0,Y 15.549,Z 391.759,A -85,B 0,C 180,E1 -31590,E2 -31590} C_VEL
LIN {X 0,Y 17.571,Z 391.592,A -85,B 0,C 180,E1 -31566.423,E2 -31566.423} C_VEL
LIN {X 0,Y 21.921,Z 390.989,A -85,B 0,C 180,E1 -31550.117,E2 -31550.117} C_VEL
LIN {X 0,Y 33.565,Z 388.524,A -85,B 0,C 180,E1 -31533.119,E2 -31533.119} C_VEL
LIN {X 0,Y 43.302,Z 385.567,A -85,B 0,C 180,E1 -31526.792,E2 -31526.792} C_VEL
LIN {X 0,Y 53.364,Z 381.576,A -85,B 0,C 180,E1 -31522.797,E2 -31522.797} C_VEL
LIN {X 0,Y 63.64,Z 376.444,A -85,B 0,C 180,E1 -31520.171,E2 -31520.171} C_VEL
LIN {X 0,Y 72.272,Z 371.183,A -85,B 0,C 180,E1 -31518.538,E2 -31518.538} C_VEL
LIN {X 0,Y 80.929,Z 364.87,A -85,B 0,C 180,E1 -31517.207,E2 -31517.207} C_VEL
LIN {X 0,Y 87.868,Z 358.925,A -85,B 0,C 180,E1 -31516.303,E2 -31516.303} C_VEL
LIN {X 0,Y 88.026,Z 358.91,A -85,B 0,C 180,E1 -31516.652,E2 -31516.652} C_VEL
LIN {X 0,Y 83.121,Z 365.656,A -85,B 0,C 180,E1 -31523.958,E2 -31523.958} C_VEL
LIN {X 0,Y 79.665,Z 371.274,A -85,B 0,C 180,E1 -31531.956,E2 -31531.956} C_VEL
LIN {X 0,Y 77.903,Z 376.343,A -85,B 0,C 180,E1 -31541.381,E2 -31541.381} C_VEL
LIN {X 0,Y 78.466,Z 380.484,A -85,B 0,C 180,E1 -31551.174,E2 -31551.174} C_VEL
LIN {X 0,Y 81.173,Z 383.52,A -85,B 0,C 180,E1 -31559.969,E2 -31559.969} C_VEL
LIN {X 0,Y 84.514,Z 385.4,A -85,B 0,C 180,E1 -31566.162,E2 -31566.162} C_VEL
LIN {X 0,Y 88.793,Z 386.824,A -85,B 0,C 180,E1 -31571.76,E2 -31571.76} C_VEL
LIN {X 0,Y 101.121,Z 388.741,A -85,B 0,C 180,E1 -31582.01,E2 -31582.01} C_VEL
LIN {X 0,Y 112.511,Z 389.144,A -85,B 0,C 180,E1 -31588.022,E2 -31588.022} C_VEL
LIN {X 0,Y 117.26,Z 389.014,A -85,B 0,C 180,E1 -31590,E2 -31590} C_VEL
LIN {X 0,Y 105.85,Z 388.97,A -85,B 0,C 180,E1 -31595.19,E2 -31595.19} C_VEL
LIN {X 0,Y 99.601,Z 388.648,A -85,B 0,C 180,E1 -31598.953,E2 -31598.953} C_VEL
LIN {X 0,Y 88.557,Z 386.753,A -85,B 0,C 180,E1 -31608.508,E2 -31608.508} C_VEL
LIN {X 0,Y 83.999,Z 385.176,A -85,B 0,C 180,E1 -31614.729,E2 -31614.729} C_VEL
LIN {X 0,Y 78.94,Z 381.288,A -85,B 0,C 180,E1 -31626.754,E2 -31626.754} C_VEL
LIN {X 0,Y 77.906,Z 376.348,A -85,B 0,C 180,E1 -31638.604,E2 -31638.604} C_VEL
LIN {X 0,Y 79.375,Z 371.965,A -85,B 0,C 180,E1 -31646.89,E2 -31646.89} C_VEL
LIN {X 0,Y 83.061,Z 365.7,A -85,B 0,C 180,E1 -31656.041,E2 -31656.041} C_VEL
LIN {X 0,Y 86.09,Z 361.606,A -85,B 0,C 180,E1 -31660.754,E2 -31660.754} C_VEL
LIN {X 0,Y 85.175,Z 362.334,A -85,B 0,C 180,E1 -31660.763,E2 -31660.763} C_VEL
LIN {X 0,Y 81.425,Z 365.959,A -85,B 0,C 180,E1 -31658.536,E2 -31658.536} C_VEL
LIN {X 0,Y 75.131,Z 372.49,A -85,B 0,C 180,E1 -31651.444,E2 -31651.444} C_VEL
LIN {X 0,Y 72.376,Z 375.919,A -85,B 0,C 180,E1 -31645.688,E2 -31645.688} C_VEL
LIN {X 0,Y 71.862,Z 376.917,A -85,B 0,C 180,E1 -31643.589,E2 -31643.589} C_VEL
LIN {X 0,Y 71.148,Z 380.747,A -85,B 0,C 180,E1 -31633.745,E2 -31633.745} C_VEL
LIN {X 0,Y 72.252,Z 383.302,A -85,B 0,C 180,E1 -31625.705,E2 -31625.705} C_VEL
LIN {X 0,Y 74.872,Z 385.451,A -85,B 0,C 180,E1 -31617.991,E2 -31617.991} C_VEL
LIN {X 0,Y 81.17,Z 387.695,A -85,B 0,C 180,E1 -31607.755,E2 -31607.755} C_VEL
LIN {X 0,Y 92.177,Z 389.128,A -85,B 0,C 180,E1 -31597.634,E2 -31597.634} C_VEL
LIN {X 0,Y 98.587,Z 389.435,A -85,B 0,C 180,E1 -31593.641,E2 -31593.641} C_VEL
LIN {X 0,Y 105.975,Z 389.318,A -85,B 0,C 180,E1 -31590,E2 -31590} C_VEL
LIN {X 0,Y 97.797,Z 389.394,A -85,B 0,C 180,E1 -31585.879,E2 -31585.879} C_VEL
LIN {X 0,Y 86.326,Z 388.559,A -85,B 0,C 180,E1 -31577.662,E2 -31577.662} C_VEL
LIN {X 0,Y 78.831,Z 387.032,A -85,B 0,C 180,E1 -31569.108,E2 -31569.108} C_VEL
LIN {X 0,Y 73.682,Z 384.681,A -85,B 0,C 180,E1 -31559.137,E2 -31559.137} C_VEL
LIN {X 0,Y 71.704,Z 382.565,A -85,B 0,C 180,E1 -31551.634,E2 -31551.634} C_VEL
LIN {X 0,Y 71.555,Z 377.746,A -85,B 0,C 180,E1 -31538.211,E2 -31538.211} C_VEL
LIN {X 0,Y 74.837,Z 372.04,A -85,B 0,C 180,E1 -31526.857,E2 -31526.857} C_VEL
LIN {X 0,Y 76.535,Z 369.835,A -85,B 0,C 180,E1 -31523.326,E2 -31523.326} C_VEL
LIN {X 0,Y 69.791,Z 374.336,A -85,B 0,C 180,E1 -31525.001,E2 -31525.001} C_VEL
LIN {X 0,Y 58.76,Z 380.319,A -85,B 0,C 180,E1 -31528.578,E2 -31528.578} C_VEL
LIN {X 0,Y 50.059,Z 384.158,A -85,B 0,C 180,E1 -31532.611,E2 -31532.611} C_VEL
LIN {X 0,Y 43.865,Z 386.527,A -85,B 0,C 180,E1 -31536.766,E2 -31536.766} C_VEL
LIN {X 0,Y 37.939,Z 388.332,A -85,B 0,C 180,E1 -31542.186,E2 -31542.186} C_VEL
LIN {X 0,Y 27.763,Z 390.797,A -85,B 0,C 180,E1 -31559.584,E2 -31559.584} C_VEL
LIN {X 0,Y 24.276,Z 391.399,A -85,B 0,C 180,E1 -31573.172,E2 -31573.172} C_VEL
LIN {X 0,Y 22.647,Z 391.567,A -85,B 0,C 180,E1 -31590,E2 -31590} C_VEL
LIN {X 0,Y 24.256,Z 391.4,A -85,B 0,C 180,E1 -31606.842,E2 -31606.842} C_VEL
LIN {X 0,Y 27.755,Z 390.797,A -85,B 0,C 180,E1 -31620.426,E2 -31620.426} C_VEL
LIN {X 0,Y 37.938,Z 388.332,A -85,B 0,C 180,E1 -31637.816,E2 -31637.816} C_VEL
LIN {X 0,Y 46.948,Z 385.374,A -85,B 0,C 180,E1 -31645.419,E2 -31645.419} C_VEL
LIN {X 0,Y 56.527,Z 381.383,A -85,B 0,C 180,E1 -31650.493,E2 -31650.493} C_VEL
LIN {X 0,Y 66.466,Z 376.25,A -85,B 0,C 180,E1 -31653.996,E2 -31653.996} C_VEL
LIN {X 0,Y 73.152,Z 372.146,A -85,B 0,C 180,E1 -31655.88,E2 -31655.88} C_VEL
LIN {X 0,Y 76.171,Z 370.305,A -85,B 0,C 180,E1 -31655.895,E2 -31655.895} C_VEL
LIN {X 0,Y 72.469,Z 375.65,A -85,B 0,C 180,E1 -31646.303,E2 -31646.303} C_VEL
LIN {X 0,Y 71.862,Z 376.917,A -85,B 0,C 180,E1 -31643.589,E2 -31643.589} C_VEL
LIN {X 0,Y 70.647,Z 379.031,A -85,B 0,C 180,E1 -31639.241,E2 -31639.241} C_VEL
LIN {X 0,Y 67.869,Z 382.439,A -85,B 0,C 180,E1 -31631.864,E2 -31631.864} C_VEL
LIN {X 0,Y 66.383,Z 385.181,A -85,B 0,C 180,E1 -31623.88,E2 -31623.88} C_VEL
LIN {X 0,Y 67.21,Z 386.299,A -85,B 0,C 180,E1 -31618.996,E2 -31618.996} C_VEL
LIN {X 0,Y 73.994,Z 388.48,A -85,B 0,C 180,E1 -31606.555,E2 -31606.555} C_VEL
LIN {X 0,Y 79.954,Z 389.319,A -85,B 0,C 180,E1 -31600.125,E2 -31600.125} C_VEL
LIN {X 0,Y 91.407,Z 389.713,A -85,B 0,C 180,E1 -31591.848,E2 -31591.848} C_VEL
LIN {X 0,Y 94.853,Z 389.619,A -85,B 0,C 180,E1 -31590,E2 -31590} C_VEL
LIN {X 0,Y 84.814,Z 389.585,A -85,B 0,C 180,E1 -31583.891,E2 -31583.891} C_VEL
LIN {X 0,Y 78.803,Z 389.242,A -85,B 0,C 180,E1 -31578.808,E2 -31578.808} C_VEL
LIN {X 0,Y 69.286,Z 387.267,A -85,B 0,C 180,E1 -31565.902,E2 -31565.902} C_VEL
LIN {X 0,Y 65.191,Z 384.736,A -85,B 0,C 180,E1 -31553.833,E2 -31553.833} C_VEL
LIN {X 0,Y 64.487,Z 381.173,A -85,B 0,C 180,E1 -31540.832,E2 -31540.832} C_VEL
LIN {X 0,Y 65.56,Z 378.915,A -85,B 0,C 180,E1 -31534.139,E2 -31534.139} C_VEL
LIN {X 0,Y 61.747,Z 380.492,A -85,B 0,C 180,E1 -31534.683,E2 -31534.683} C_VEL
LIN {X 0,Y 54.227,Z 383.966,A -85,B 0,C 180,E1 -31538.958,E2 -31538.958} C_VEL
LIN {X 0,Y 48.478,Z 386.334,A -85,B 0,C 180,E1 -31543.544,E2 -31543.544} C_VEL
LIN {X 0,Y 43.055,Z 388.139,A -85,B 0,C 180,E1 -31549.238,E2 -31549.238} C_VEL
LIN {X 0,Y 34.108,Z 390.605,A -85,B 0,C 180,E1 -31565.663,E2 -31565.663} C_VEL
LIN {X 0,Y 31.161,Z 391.207,A -85,B 0,C 180,E1 -31576.966,E2 -31576.966} C_VEL
LIN {X 0,Y 29.763,Z 391.375,A -85,B 0,C 180,E1 -31590,E2 -31590} C_VEL
LIN {X 0,Y 31.143,Z 391.208,A -85,B 0,C 180,E1 -31603.042,E2 -31603.042} C_VEL
LIN {X 0,Y 34.1,Z 390.605,A -85,B 0,C 180,E1 -31614.342,E2 -31614.342} C_VEL
LIN {X 0,Y 43.054,Z 388.139,A -85,B 0,C 180,E1 -31630.763,E2 -31630.763} C_VEL
LIN {X 0,Y 51.325,Z 385.182,A -85,B 0,C 180,E1 -31638.861,E2 -31638.861} C_VEL
LIN {X 0,Y 60.363,Z 381.19,A -85,B 0,C 180,E1 -31644.587,E2 -31644.587} C_VEL
LIN {X 0,Y 61.39,Z 380.683,A -85,B 0,C 180,E1 -31645.087,E2 -31645.087} C_VEL
LIN {X 0,Y 65.572,Z 378.912,A -85,B 0,C 180,E1 -31645.858,E2 -31645.858} C_VEL
LIN {X 0,Y 64.346,Z 382.502,A -85,B 0,C 180,E1 -31634.981,E2 -31634.981} C_VEL
LIN {X 0,Y 66.245,Z 385.745,A -85,B 0,C 180,E1 -31621.933,E2 -31621.933} C_VEL
LIN {X 0,Y 67.21,Z 386.299,A -85,B 0,C 180,E1 -31618.996,E2 -31618.996} C_VEL
LIN {X 0,Y 68.554,Z 387.366,A -85,B 0,C 180,E1 -31614.199,E2 -31614.199} C_VEL
LIN {X 0,Y 70.205,Z 388.825,A -85,B 0,C 180,E1 -31606.201,E2 -31606.201} C_VEL
LIN {X 0,Y 72.43,Z 389.628,A -85,B 0,C 180,E1 -31600.133,E2 -31600.133} C_VEL
LIN {X 0,Y 75.326,Z 389.924,A -85,B 0,C 180,E1 -31596.169,E2 -31596.169} C_VEL
LIN {X 0,Y 76.586,Z 389.992,A -85,B 0,C 180,E1 -31595.037,E2 -31595.037} C_VEL
LIN {X 0,Y 83.889,Z 389.915,A -85,B 0,C 180,E1 -31590,E2 -31590} C_VEL
LIN {X 0,Y 76.28,Z 389.976,A -85,B 0,C 180,E1 -31584.714,E2 -31584.714} C_VEL
LIN {X 0,Y 65.944,Z 389.092,A -85,B 0,C 180,E1 -31573.561,E2 -31573.561} C_VEL
LIN {X 0,Y 60.324,Z 387.579,A -85,B 0,C 180,E1 -31562.224,E2 -31562.224} C_VEL
LIN {X 0,Y 57.526,Z 384.791,A -85,B 0,C 180,E1 -31547.135,E2 -31547.135} C_VEL
LIN {X 0,Y 53.644,Z 386.142,A -85,B 0,C 180,E1 -31549.077,E2 -31549.077} C_VEL
LIN {X 0,Y 48.679,Z 387.947,A -85,B 0,C 180,E1 -31554.725,E2 -31554.725} C_VEL
LIN {X 0,Y 40.728,Z 390.412,A -85,B 0,C 180,E1 -31569.811,E2 -31569.811} C_VEL
LIN {X 0,Y 38.125,Z 391.015,A -85,B 0,C 180,E1 -31579.377,E2 -31579.377} C_VEL
LIN {X 0,Y 36.867,Z 391.184,A -85,B 0,C 180,E1 -31590,E2 -31590} C_VEL
LIN {X 0,Y 38.11,Z 391.015,A -85,B 0,C 180,E1 -31600.627,E2 -31600.627} C_VEL
LIN {X 0,Y 40.701,Z 390.412,A -85,B 0,C 180,E1 -31610.203,E2 -31610.203} C_VEL
LIN {X 0,Y 48.678,Z 387.947,A -85,B 0,C 180,E1 -31625.275,E2 -31625.275} C_VEL
LIN {X 0,Y 53.646,Z 386.142,A -85,B 0,C 180,E1 -31630.922,E2 -31630.922} C_VEL
LIN {X 0,Y 57.543,Z 384.782,A -85,B 0,C 180,E1 -31632.883,E2 -31632.883} C_VEL
LIN {X 0,Y 60.354,Z 387.578,A -85,B 0,C 180,E1 -31617.761,E2 -31617.761} C_VEL
LIN {X 0,Y 69.623,Z 389.603,A -85,B 0,C 180,E1 -31601.647,E2 -31601.647} C_VEL
LIN {X 0,Y 76.586,Z 389.992,A -85,B 0,C 180,E1 -31595.037,E2 -31595.037} C_VEL
LIN {X 0,Y 77.13,Z 390.085,A -85,B 0,C 180,E1 -31593.77,E2 -31593.77} C_VEL
LIN {X 0,Y 76.499,Z 390.146,A -85,B 0,C 180,E1 -31591.981,E2 -31591.981} C_VEL
LIN {X 0,Y 74.295,Z 390.232,A -85,B 0,C 180,E1 -31589.609,E2 -31589.609} C_VEL
LIN {X 0,Y 63.335,Z 390.124,A -85,B 0,C 180,E1 -31581.287,E2 -31581.287} C_VEL
LIN {X 0,Y 58.365,Z 389.764,A -85,B 0,C 180,E1 -31574.418,E2 -31574.418} C_VEL
LIN {X 0,Y 53.336,Z 388.635,A -85,B 0,C 180,E1 -31563.363,E2 -31563.363} C_VEL
LIN {X 0,Y 50.745,Z 389.148,A -85,B 0,C 180,E1 -31565.45,E2 -31565.45} C_VEL
LIN {X 0,Y 47.498,Z 390.219,A -85,B 0,C 180,E1 -31572.787,E2 -31572.787} C_VEL
LIN {X 0,Y 45.148,Z 390.823,A -85,B 0,C 180,E1 -31581.045,E2 -31581.045} C_VEL
LIN {X 0,Y 43.963,Z 390.992,A -85,B 0,C 180,E1 -31590,E2 -31590} C_VEL
LIN {X 0,Y 45.116,Z 390.824,A -85,B 0,C 180,E1 -31598.962,E2 -31598.962} C_VEL
LIN {X 0,Y 47.473,Z 390.219,A -85,B 0,C 180,E1 -31607.222,E2 -31607.222} C_VEL
LIN {X 0,Y 50.74,Z 389.149,A -85,B 0,C 180,E1 -31614.552,E2 -31614.552} C_VEL
LIN {X 0,Y 53.346,Z 388.63,A -85,B 0,C 180,E1 -31616.665,E2 -31616.665} C_VEL
LIN {X 0,Y 59.588,Z 389.88,A -85,B 0,C 180,E1 -31603.644,E2 -31603.644} C_VEL
LIN {X 0,Y 71.591,Z 390.247,A -85,B 0,C 180,E1 -31591.151,E2 -31591.151} C_VEL
LIN {X 0,Y 73.187,Z 390.203,A -85,B 0,C 180,E1 -31590,E2 -31590} C_VEL
LIN {X 0,Y 63.335,Z 390.124,A -85,B 0,C 180,E1 -31581.287,E2 -31581.287} C_VEL
LIN {X 0,Y 61.447,Z 390.129,A -85,B 0,C 180,E1 -31580.359,E2 -31580.359} C_VEL
LIN {X 0,Y 58.196,Z 390.293,A -85,B 0,C 180,E1 -31580.648,E2 -31580.648} C_VEL
LIN {X 0,Y 54.603,Z 390.576,A -85,B 0,C 180,E1 -31582.711,E2 -31582.711} C_VEL
LIN {X 0,Y 52.377,Z 390.769,A -85,B 0,C 180,E1 -31585.271,E2 -31585.271} C_VEL
LIN {X 0,Y 51.22,Z 390.769,A -85,B 0,C 180,E1 -31588.575,E2 -31588.575} C_VEL
LIN {X 0,Y 51.086,Z 390.8,A -85,B 0,C 180,E1 -31590,E2 -31590} C_VEL
LIN {X 0,Y 52.182,Z 390.631,A -85,B 0,C 180,E1 -31597.74,E2 -31597.74} C_VEL
LIN {X 0,Y 54.073,Z 390.454,A -85,B 0,C 180,E1 -31599.165,E2 -31599.165} C_VEL
LIN {X 0,Y 62.614,Z 390.489,A -85,B 0,C 180,E1 -31590,E2 -31590} C_VEL
LIN {X 0,Y 54.082,Z 390.456,A -85,B 0,C 180,E1 -31580.858,E2 -31580.858} C_VEL
LIN {X 0,Y 52.214,Z 390.63,A -85,B 0,C 180,E1 -31582.265,E2 -31582.265} C_VEL
LIN {X 0,Y 51.22,Z 390.769,A -85,B 0,C 180,E1 -31588.575,E2 -31588.575} C_VEL
LIN {X 0,Y 51.028,Z 392.768,A -85,B 0,C 180,E1 -31590.752,E2 -31590.752} C_VEL
LIN {X 0,Y 51.028,Z 600,A -85,B 0,C 180,E1 -31590.752,E2 -31590.752} C_VEL
LIN {X 0,Y 51.028,Z 600,A -85,B 0,C 180,E1 -31590.752,E2 -31590.752}

QRS_NEXT_CUT()

QRS_NEXT()
QRS_HOME()

END
